// TwinCAT 3 PLC project Proxy
// ProgramVersion: 3.1.4023.0
// libraries:
//   Tc2_Standard, * (Beckhoff Automation GmbH)
//   Tc2_System, * (Beckhoff Automation GmbH)
//   Tc3_Module, * (Beckhoff Automation GmbH)
// project tree:
//   / Class Diagram_Proxy.TcCD (not stored), PlcTask.TcTTO
//   Classes/ Proxy.TcPOU, Realsubject.TcPOU
//   GVLs/ GVL.TcGVL
//   Interfaces/ Subject_Interface.TcIO
//   POUs/ MAIN.TcPOU, PLC_PRG.TcPOU
// real-time tasks:
//   TASK PlcTask: cycle T#10ms, priority 20, ADS port 350

CONFIGURATION Proxy
    RESOURCE PLC ON TwinCAT3
        TASK PlcTask(INTERVAL := T#10ms, PRIORITY := 20);
        PROGRAM MAIN WITH PlcTask : MAIN;
    END_RESOURCE
END_CONFIGURATION

// ---- GVLs/GVL.TcGVL
{attribute 'qualified_only' := ''}
VAR_GLOBAL
	///Realsubject class instance
	globalSubjectInstance: Realsubject;
END_VAR

// ---- Interfaces/Subject_Interface.TcIO
INTERFACE Subject_Interface

METHOD Get_Method : INT
END_METHOD

METHOD Set_Method
VAR_INPUT
	///Value to be set passed as an argument
	num: INT;
END_VAR
END_METHOD

END_INTERFACE

// ---- POUs/MAIN.TcPOU
PROGRAM MAIN
VAR
END_VAR

PLC_PRG();

END_PROGRAM

// ---- POUs/PLC_PRG.TcPOU
PROGRAM PLC_PRG
VAR
	///Instance of Realsubject but this one is Local to prove on a local and a global object
	localSubjectInstance: Realsubject;
	///Pointer to the local subject. Needed to instantiate its own Proxy. 
	ptrLocalSubject: POINTER TO Realsubject := ADR(localSubjectInstance);
	///Null pointer to the RealSubject class to verify that the other pointers are valid pointers and not null
	ptrNullRealSubject: POINTER TO Realsubject;
	///Pointer needed to create the Connection bridge "Proxy" between the client and the subject 
	ptrProxy: POINTER TO Proxy;
	///Variable to store the password set by the client to perform the connection
	iTempPasswordLocal: INT;
	///Variable to store the INT passed by the client to be SET on the subject
	iSetValueLocal: INT;
	///Boolean value to that gets toggled when the client send a SET request.
	///It is toggled again after the Proxy's response
	bWriteRequest: BOOL;
	///Boolean value to that gets toggled when the client send a GET request.
	///It is toggled again after the Proxy's response
	bReadRequest: BOOL;
	///Variable to store locally if the request was a Write or Read request.
	///TRUE for a Write request and FALSE for a Read request
	bReadWriteLocal: BOOL;
END_VAR
VAR_INPUT
	///Variable to store the response log from the Proxy on a SET request
	sTempSetLog: STRING := 'Waiting for a request';
	///Variable to store the response log from the Proxy on a GET request
	sTempGetLog: STRING := 'Waiting for a request';
	///Variable to store the LAST GET response value locally
	iGetValueLocal: INT;
END_VAR

//The Visualization element can send a GET/SET request with all its parameters.
//Once the request is received by the PLC_PRG, the PLC_PRG creates the Proxy object to delegate the request and subject's connection to it.
//The default password value for the request is: 1234. It is specified in the static field .iRealPassword of the Proxy class

//El elemento Visualización puede enviar una solicitud GET/SET con todos sus parámetros.
// Una vez que PLC_PRG recibe la solicitud, PLC_PRG crea el objeto Proxy para delegar la solicitud y la conexión del sujeto a ella.
//El valor de contraseña predeterminado para la solicitud es: 1234. Se especifica en el campo estático .iRealPassword de la clase Proxy

//If a WRITE or SET request is received
IF	bWriteRequest THEN
	
	//We specify TRUE bReadWriteLocal because it is a SET request
	bReadWriteLocal := TRUE;
	//First we verify if the pointer to RealSubject to be used is a valid pointer
	IF ptrLocalSubject <> ptrNullRealSubject THEN
		//If so, 
		
		//The Proxy object is created with all its parameters passed by the PLC_PRG local variables.
		//As there is no "Method Overloading" options is CODESYS (Or at least the constructor cannot be overloaded) the constructor must receive and handle all the possible scenarios
		// .ptrToRealSubject is a Pointer to the RealSubject instance that we try to conncect to
		// .iTempPassword is the password passed by the client in the visualization element
		// .iSetValue is the value passed by the client to be SET on the RealSubject. If the request is a GET request, this value has no effect on the output of the connection.
		// .bReadWrite is the boolean value that specifies if the request is a SET or GET request
		
		//El objeto Proxy se crea con todos sus parámetros pasados ​​por las variables locales PLC_PRG.
		//Como no hay opciones de "Sobrecarga de métodos" en CODESYS (O al menos el constructor no se puede sobrecargar) el constructor debe recibir y manejar todos los escenarios posibles
		// .ptrToRealSubject es un puntero a la instancia de RealSubject a la que intentamos conectarnos
		// .iTempPassword es la contraseña pasada por el cliente en el elemento de visualización
		// .iSetValue es el valor pasado por el cliente para establecerlo en RealSubject. Si la solicitud es una solicitud GET, este valor no tiene ningún efecto en la salida de la conexión.
		// .bReadWrite es el valor booleano que especifica si la solicitud es una solicitud SET o GET		
		
		ptrProxy := __NEW( Proxy( ptrToRealSubject := ptrLocalSubject, iTempPassword :=  iTempPasswordLocal, iSetValue := iSetValueLocal, bReadWrite := bReadWriteLocal));
		//Once the Proxy has made the response, the memory is released by deleting the Proxy object
		__DELETE(ptrProxy);
	END_IF
	
	//We delete the local value of last password for security reasons. This way for every request the client must input a password
	iTempPasswordLocal := 0;
	//Once the WRITE request has been handled, we toggle the variable to avoid double requests
	bWriteRequest := FALSE;
END_IF

//If a READ or GET request is received
IF	bReadRequest THEN
	
	//We specify FALSE bReadWriteLocal because it is a GET request
	bReadWriteLocal := FALSE;
	//First we verify if the pointer to RealSubject to be used is a valid pointer
	IF ptrLocalSubject <> ptrNullRealSubject THEN
		//If so,
		
		//The Proxy object is created with all its parameters passed by the PLC_PRG local variables.
		//As there is no "Method Overloading" options is CODESYS (Or at least the constructor cannot be overloaded) the constructor must receive and handle all the possible scenarios
		// .ptrToRealSubject is a Pointer to the RealSubject instance that we try to conncect to
		// .iTempPassword is the password passed by the client in the visualization element
		// .iSetValue is the value passed by the client to be SET on the RealSubject. If the request is a GET request, this value has no effect on the output of the connection.
		// .bReadWrite is the boolean value that specifies if the request is a SET or GET request
		
		//El objeto Proxy se crea con todos sus parámetros pasados ​​por las variables locales PLC_PRG.
		//Como no hay opciones de "Sobrecarga de métodos" en CODESYS (O al menos el constructor no se puede sobrecargar) el constructor debe recibir y manejar todos los escenarios posibles
		// .ptrToRealSubject es un puntero a la instancia de RealSubject a la que intentamos conectarnos
		// .iTempPassword es la contraseña pasada por el cliente en el elemento de visualización
		// .iSetValue es el valor pasado por el cliente para establecerlo en RealSubject. Si la solicitud es una solicitud GET, este valor no tiene ningún efecto en la salida de la conexión.
		// .bReadWrite es el valor booleano que especifica si la solicitud es una solicitud SET o GET
		
		ptrProxy := __NEW(Proxy(ptrToRealSubject := ptrLocalSubject, iTempPassword :=  iTempPasswordLocal, iSetValue := 0, bReadWrite := bReadWriteLocal));
		//Once the Proxy has made the response, the memory is released by deleting the Proxy object
		__DELETE(ptrProxy);	
	END_IF
	
	//We delete the local value of last password for security reasons. This way for every request the client must input a password
	iTempPasswordLocal := 0;
	//Once the READ request has been handled, we toggle the variable to avoid double requests
	bReadRequest := FALSE;
END_IF

END_PROGRAM

// ---- Classes/Realsubject.TcPOU
{attribute 'enable_dynamic_creation' := ''}
FUNCTION_BLOCK Realsubject IMPLEMENTS Subject_Interface
VAR
	///Variable to get and set values
	iProp: INT;
END_VAR

METHOD Get_Method : INT
//Asks for the value of the object's iProp variable and passes it to the caller

Get_Method := THIS^.iProp;
END_METHOD

METHOD Set_Method
VAR_INPUT
	///Value to be set on the iProp varible of realSubjectInstance
	num: INT;
END_VAR
//Stores the value of the caller object on iProp variable. 

THIS^.iProp := num;
END_METHOD

END_FUNCTION_BLOCK

// ---- Classes/Proxy.TcPOU
{attribute 'enable_dynamic_creation' := ''}
FUNCTION_BLOCK Proxy IMPLEMENTS Subject_Interface
VAR
	///Pointer to store the reference to the subject being protected
	refToRealSubject: POINTER TO Realsubject;
	///Last value of password entered by the client in the visualization element
	iTempPassword: INT;
END_VAR
VAR_STAT
	///Default password value for the request to be accepted
	iRealPassword: INT := 1234;
END_VAR

METHOD fb_init
VAR_INPUT
	/// TRUE: the Retain-variables are initialized (reset warm / reset cold)
	bInitRetains: BOOL;
	/// TRUE  the instance will be copied to the copy-code afterward (online change)
	bInCopyCode: BOOL;
	///Pointer to the RealSubject instance 
	ptrToRealSubject: POINTER TO Realsubject;
	///Local variable to store the password passed by the client with the password of the Proxy
	iTempPassword: INT;
	///Local variable to be used in WRITE request, it is the value to be set if the request is accepted
	iSetValue: INT;
	///Boolean value that specifies if the request is a WRITE or READ request
	bReadWrite: BOOL;
END_VAR
//Stores the address of the subject on a field in th Proxy.
THIS^.refToRealSubject := ptrToRealSubject;
//Stores the password value of the client on a field in the Proxy
THIS^.iTempPassword := iTempPassword;

//For security reasons, the Password passed by the client and the Proxi's connection password are compared
IF	THIS^.iTempPassword = THIS^.iRealPassword THEN
	//If the password sent by the client is correct,
	
	//We verify is the request is a SET or GET request
	IF bReadWrite THEN
		//If the request is a SET request: boolean value TRUE
		
		//The Proxy passes the request to the subject
		THIS^.Set_Method(iSetValue);
		//Once the request is completed, the Proxy responds to the client that the request has been accepted
		PLC_PRG.sTempSetLog := 'Request "SET" accepted';
		//If the request is a GET request: boolean value FALSE
	ELSE
		//The Proxy passes the request to the subject
		PLC_PRG.iGetValueLocal:= THIS^.Get_Method();
		//Once the request is completed, the Proxy responds to the client that the request has been accepted
		PLC_PRG.sTempGetLog := 'Request "GET" accepted';
	END_IF
	
	//If the password sent by the client is incorrect
ELSE 
	//We verify is the request is a SET or GET request
	IF bReadWrite THEN
		//If the request is a SET request: boolean value TRUE
		
		//The Proxy handles the bad request and response to the client without the subject intervention
		PLC_PRG.sTempSetLog := 'Request denied. Wrong password.';
		//If the request is a GET request: boolean value FALSE
	ELSE
		//The Proxy handles the bad request and response to the client without the subject intervention
		PLC_PRG.sTempGetLog := 'Request denied. Wrong password.';
	END_IF

END_IF
END_METHOD

METHOD Get_Method : INT
//Calls the Get_Method of the subject through the proxy to read the iProp value of the subject 
// thanks to the pointer reference saved in the field refToRealSubject of the proxy object. 

Get_Method := THIS^.refToRealSubject^.Get_Method();
END_METHOD

METHOD Set_Method
VAR_INPUT
	///Value to be set to the subject passed as an input argument
	num: INT;
END_VAR
//Calls the Set_Method of the subject through the proxy to write the iProp field of the subject 
// thanks to the pointer reference saved in the field refToRealSubject of the proxy object.

THIS^.refToRealSubject^.Set_Method(num);
END_METHOD

END_FUNCTION_BLOCK
